PROGRAM P1_04_MachineControl
VAR
	tonStarting		:TON;
	tonStopping		:TON;
	
	
	
	
	doorunlocked: INT;
	tofDoorLocked: TOF;
END_VAR

VAR PERSISTENT
	bBatchConfirmation1			:BOOL;
	bBatchConfirmation2			:BOOL;
	bBatchConfirmation3			:BOOL;
	bBatchConfirmation4			:BOOL;
END_VAR
VAR // added by the converter: edge detectors and wires of the graphical bodies
    _w1, _w2, _w3, _w4, _w5, _w6, _w7, _w8 : BOOL;
    _ft1 : F_TRIG;
    _rt1, _rt2 : R_TRIG;
END_VAR

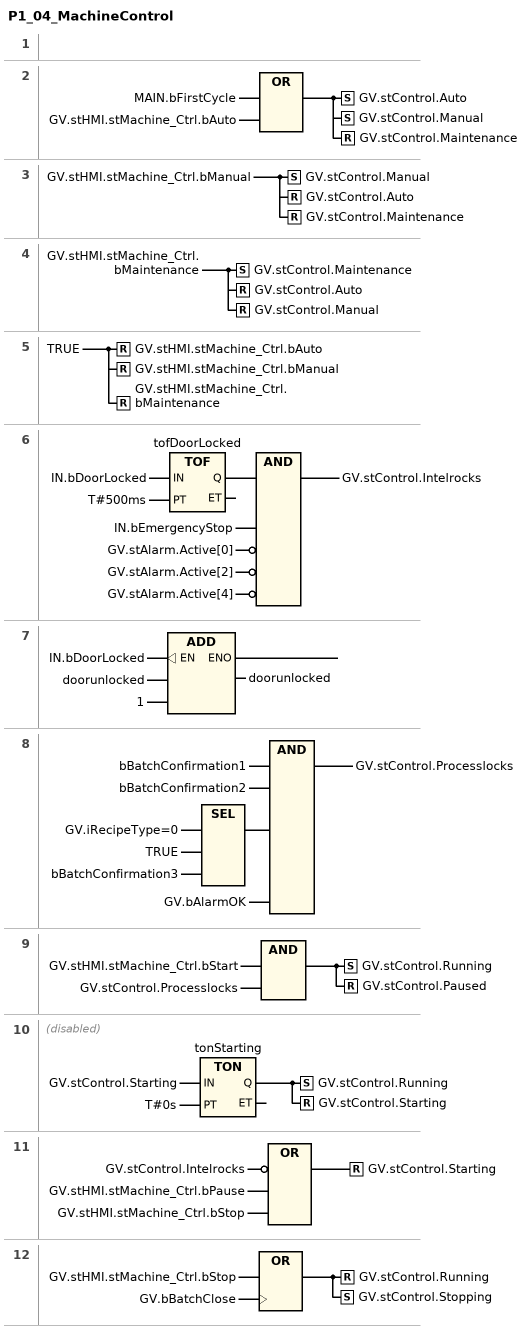
// NETWORK 1

// NETWORK 2
_w1 := MAIN.bFirstCycle OR GV.stHMI.stMachine_Ctrl.bAuto;
GV.stControl.Auto S= _w1;
GV.stControl.Manual S= _w1;
GV.stControl.Maintenance R= _w1;

// NETWORK 3
_w2 := GV.stHMI.stMachine_Ctrl.bManual;
GV.stControl.Manual S= _w2;
GV.stControl.Auto R= _w2;
GV.stControl.Maintenance R= _w2;

// NETWORK 4
_w3 := GV.stHMI.stMachine_Ctrl.bMaintenance;
GV.stControl.Maintenance S= _w3;
GV.stControl.Auto R= _w3;
GV.stControl.Manual R= _w3;

// NETWORK 5
GV.stHMI.stMachine_Ctrl.bAuto R= TRUE;
GV.stHMI.stMachine_Ctrl.bManual R= TRUE;
GV.stHMI.stMachine_Ctrl.bMaintenance R= TRUE;

// NETWORK 6
tofDoorLocked(IN := IN.bDoorLocked, PT := T#500ms); // TOF
GV.stControl.Intelrocks := tofDoorLocked.Q AND IN.bEmergencyStop AND NOT GV.stAlarm.Active[0] AND NOT GV.stAlarm.Active[2] AND NOT GV.stAlarm.Active[4];

// NETWORK 7
_ft1(CLK := IN.bDoorLocked);
IF _ft1.Q THEN doorunlocked := doorunlocked + 1; END_IF

// NETWORK 8
GV.stControl.Processlocks := bBatchConfirmation1 AND bBatchConfirmation2 AND SEL(GV.iRecipeType=0, TRUE, bBatchConfirmation3) AND GV.bAlarmOK;

// NETWORK 9
_w4 := GV.stHMI.stMachine_Ctrl.bStart AND GV.stControl.Processlocks;
GV.stControl.Running S= _w4;
GV.stControl.Paused R= _w4;

// NETWORK 10 (disabled)
// tonStarting(IN := GV.stControl.Starting, PT := T#0s); // TON
// GV.stControl.Running S= tonStarting.Q;
// GV.stControl.Starting R= tonStarting.Q;

// NETWORK 11
GV.stControl.Starting R= NOT GV.stControl.Intelrocks OR GV.stHMI.stMachine_Ctrl.bPause OR GV.stHMI.stMachine_Ctrl.bStop;

// NETWORK 12
_rt1(CLK := GV.bBatchClose);
_w5 := GV.stHMI.stMachine_Ctrl.bStop OR _rt1.Q;
GV.stControl.Running R= _w5;
GV.stControl.Stopping S= _w5;

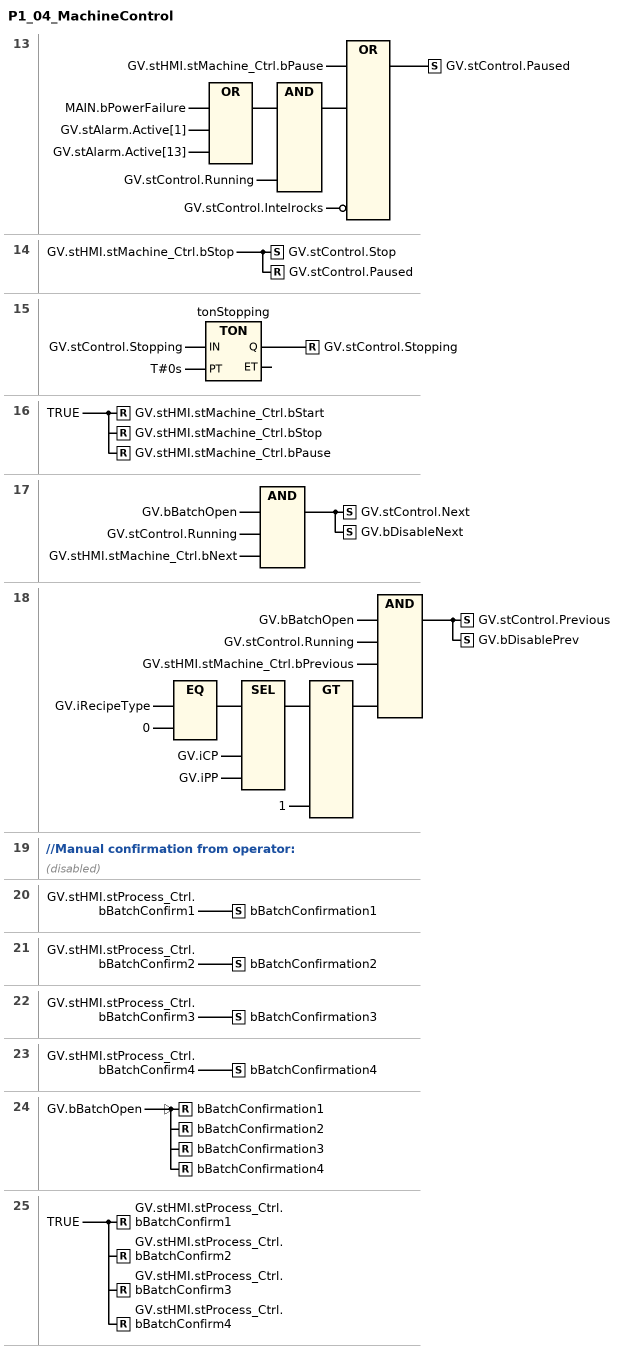
// NETWORK 13
GV.stControl.Paused S= GV.stHMI.stMachine_Ctrl.bPause OR (MAIN.bPowerFailure OR GV.stAlarm.Active[1] OR GV.stAlarm.Active[13]) AND GV.stControl.Running OR NOT GV.stControl.Intelrocks;

// NETWORK 14
_w6 := GV.stHMI.stMachine_Ctrl.bStop;
GV.stControl.Stop S= _w6;
GV.stControl.Paused R= _w6;

// NETWORK 15
tonStopping(IN := GV.stControl.Stopping, PT := T#0s); // TON
GV.stControl.Stopping R= tonStopping.Q;

// NETWORK 16
GV.stHMI.stMachine_Ctrl.bStart R= TRUE;
GV.stHMI.stMachine_Ctrl.bStop R= TRUE;
GV.stHMI.stMachine_Ctrl.bPause R= TRUE;

// NETWORK 17
_w7 := GV.bBatchOpen AND GV.stControl.Running AND GV.stHMI.stMachine_Ctrl.bNext;
GV.stControl.Next S= _w7;
GV.bDisableNext S= _w7;

// NETWORK 18
_w8 := GV.bBatchOpen AND GV.stControl.Running AND GV.stHMI.stMachine_Ctrl.bPrevious AND SEL(GV.iRecipeType = 0, GV.iCP, GV.iPP) > 1;
GV.stControl.Previous S= _w8;
GV.bDisablePrev S= _w8;

// NETWORK 19 (disabled)
// label: //Manual confirmation from operator

// NETWORK 20
bBatchConfirmation1 S= GV.stHMI.stProcess_Ctrl.bBatchConfirm1;

// NETWORK 21
bBatchConfirmation2 S= GV.stHMI.stProcess_Ctrl.bBatchConfirm2;

// NETWORK 22
bBatchConfirmation3 S= GV.stHMI.stProcess_Ctrl.bBatchConfirm3;

// NETWORK 23
bBatchConfirmation4 S= GV.stHMI.stProcess_Ctrl.bBatchConfirm4;

// NETWORK 24
_rt2(CLK := GV.bBatchOpen);
bBatchConfirmation1 R= _rt2.Q;
bBatchConfirmation2 R= _rt2.Q;
bBatchConfirmation3 R= _rt2.Q;
bBatchConfirmation4 R= _rt2.Q;

// NETWORK 25
GV.stHMI.stProcess_Ctrl.bBatchConfirm1 R= TRUE;
GV.stHMI.stProcess_Ctrl.bBatchConfirm2 R= TRUE;
GV.stHMI.stProcess_Ctrl.bBatchConfirm3 R= TRUE;
GV.stHMI.stProcess_Ctrl.bBatchConfirm4 R= TRUE;

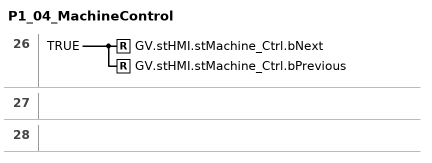
// NETWORK 26
GV.stHMI.stMachine_Ctrl.bNext R= TRUE;
GV.stHMI.stMachine_Ctrl.bPrevious R= TRUE;

// NETWORK 27

// NETWORK 28

END_PROGRAM

(* stored: Version 1.1.0.1
   POU P1_04_MachineControl: Id {28291006-7217-4dfd-bae8-40d23c5c0960}, SpecialFunc None *)
